FUNCTION_BLOCK Coordinator
  (* Version 1.0, 2006-11-13, Goran Cengic, Chalmers *)
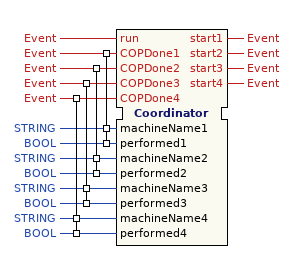
  EVENT_INPUT
    run;
    COPDone1 WITH machineName1, performed1;
    COPDone2 WITH machineName2, performed2;
    COPDone3 WITH machineName3, performed3;
    COPDone4 WITH machineName4, performed4;
  END_EVENT
  EVENT_OUTPUT
    start1;
    start2;
    start3;
    start4;
  END_EVENT
  VAR_INPUT
    machineName1 : STRING;
    performed1 : BOOL;
    machineName2 : STRING;
    performed2 : BOOL;
    machineName3 : STRING;
    performed3 : BOOL;
    machineName4 : STRING;
    performed4 : BOOL;
  END_VAR
END_FUNCTION_BLOCK
